VISUALIZATION VAC  // 2x2
END_VISUALIZATION

(* stored: Version 1.1.0.1, ProductVersion 3.1.0.26
   Visu VAC: Id {4fe33960-aa3a-4b8f-8b92-3308e23ba822} *)
